TYPE ST_safetyDoor :
STRUCT
	button_reset		: BOOL;
	button_unlock		: BOOL;
	button_lock			: BOOL;
	door_closed			: BOOL;
	door_locked			: BOOL;
	
	lamp_reset			: BOOL;
	lamp_unlock			: BOOL;
	lamp_lock			: BOOL;
	door_lock			: BOOL;
END_STRUCT
END_TYPE

(* stored: Version 1.1.0.1, ProductVersion 3.1.4024.12
   DUT ST_safetyDoor: Id {35b1bffa-3fd7-4efb-8bb2-e8e5f76ef9f1} *)
